FUNCTION_BLOCK WTAV_PCT (* Percent Weighted Average *)
  (* Standard: 61499-1; Classification: Math; Function: Weighted average; Type: Percent *)
  (* Version 0.0, 2006-04-07, JHC, Holobloc Inc, Derived from WTAV_UINT. *)
  (* Compiler header: package fb.rt.math; *)
  (* Compiler Java Sun JDK 1.5.0 *)
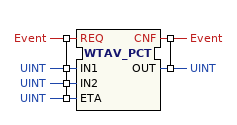
  EVENT_INPUT
    REQ WITH IN1, IN2, ETA; (* Normal Calculation *)
  END_EVENT
  EVENT_OUTPUT
    CNF WITH OUT; (* Execution Confirmation *)
  END_EVENT
  VAR_INPUT
    IN1 : UINT; (* Value when ETA=0 *)
    IN2 : UINT; (* Value when ETA=100 *)
    ETA : UINT; (* Weighting factor, percent *)
  END_VAR
  VAR_OUTPUT
    OUT : UINT; (* ETA*X1+(1-ETA)*X2 *)
  END_VAR
  ALGORITHM REQ IN ST: (* Normally executed algorithm *)
OUT := ((100-ETA)*IN1 + ETA*IN2)/100;
CNF.serviceEvent(this);
  END_ALGORITHM
END_FUNCTION_BLOCK
